# EPICS IOC start-up script: compress/start.iocsh
require calc, 3.7.3
dbLoadTemplate("comp_ex1.substitution")
